(* IEC 61131-3 sources: plc/src/scl/function_blocks, 4 files *)

(* ---- dol_starter.fb ---- *)
FUNCTION_BLOCK FB DOL_Starter
VAR_INPUT
    // Digital inputs
    bStart_PB : BOOL;         // Start push button (NO)
    bStop_PB : BOOL;          // Stop push button (NC - active when pressed)
    bOverload : BOOL;         // Overload relay contact (NC - active when tripped)
    bAux_Contact : BOOL;      // Contactor auxiliary feedback (NO)
END_VAR

VAR_OUTPUT
    // Digital outputs
    bContactor : BOOL;        // Contactor coil output
    bRunning_Ind : BOOL;      // Motor running indicator
    bFault_Ind : BOOL;        // Fault indicator
    bReady_Ind : BOOL;        // Ready status indicator
END_VAR

VAR
    // Internal variables
    bLatching : BOOL;         // Latching signal
    bFault_Memory : BOOL;     // Fault memory (requires reset)
    bStart_Memory : BOOL;     // Start command memory
    bStop_Memory : BOOL;      // Stop command memory
    tStart_Delay : TON;       // Start delay timer
    tFault_Delay : TON;       // Fault delay timer
END_VAR

BEGIN
    // ==========================================
    // DOL Starter Main Control Logic
    // ==========================================

    // Input signal conditioning with debouncing
    // Rising edge detection for start button
    IF bStart_PB AND NOT bStart_Memory THEN
        bStart_Memory := TRUE;
    ELSIF NOT bStart_PB THEN
        bStart_Memory := FALSE;
    END_IF;

    // Rising edge detection for stop button (inverted - active when pressed)
    IF bStop_PB AND NOT bStop_Memory THEN
        bStop_Memory := TRUE;
    ELSIF NOT bStop_PB THEN
        bStop_Memory := FALSE;
    END_IF;

    // ==========================================
    // Main Control Circuit (Network 1 equivalent)
    // ==========================================

    // Start condition: Start button pressed AND no stop AND no overload AND no fault
    IF bStart_PB AND NOT bStop_PB AND NOT bOverload AND NOT bFault_Memory THEN
        bLatching := TRUE;
    END_IF;

    // Stop conditions: Stop button pressed OR overload OR fault
    IF bStop_PB OR bOverload OR bFault_Memory THEN
        bLatching := FALSE;
    END_IF;

    // Fault memory setting (latches fault condition)
    IF bOverload THEN
        bFault_Memory := TRUE;
    END_IF;

    // ==========================================
    // Contactor Control
    // ==========================================

    // Contactor output with latching
    // Start delay for smooth starting (optional)
    tStart_Delay(IN := bLatching, PT := T#100MS);

    bContactor := tStart_Delay.Q AND NOT bFault_Memory;

    // ==========================================
    // Status Indication (Networks 2-4 equivalent)
    // ==========================================

    // Running indicator (Network 2)
    bRunning_Ind := bContactor AND bAux_Contact;

    // Fault indicator (Network 3)
    bFault_Ind := bFault_Memory OR bOverload;

    // Ready indicator (Network 4)
    bReady_Ind := NOT bStop_PB AND NOT bOverload AND NOT bFault_Memory AND NOT bContactor;

    // ==========================================
    // Additional Safety Features
    // ==========================================

    // Contactor feedback monitoring
    // If contactor output is ON but auxiliary feedback is OFF, indicate fault
    IF bContactor AND NOT bAux_Contact THEN
        tFault_Delay(IN := TRUE, PT := T#500MS);
        IF tFault_Delay.Q THEN
            bFault_Memory := TRUE; // Contactor fault
        END_IF;
    ELSE
        tFault_Delay(IN := FALSE);
    END_IF;

    // Auto-reset fault memory when conditions are safe
    // (Optional - remove if manual reset is preferred)
    IF NOT bOverload AND NOT bContactor AND bStop_PB THEN
        // Fault can be reset by pressing stop button when safe
        bFault_Memory := FALSE;
    END_IF;

END_FUNCTION_BLOCK

(* ---- dol_starter_s7_1500.fb ---- *)
FUNCTION_BLOCK FB DOL_Starter_S7_1500
{ S7_Optimized_Access := 'TRUE' }
VAR_INPUT
    // Digital inputs
    bStart_PB : BOOL;         // Start push button (NO)
    bStop_PB : BOOL;          // Stop push button (NC - active when pressed)
    bOverload : BOOL;         // Overload relay contact (NC - active when tripped)
    bAux_Contact : BOOL;      // Contactor auxiliary feedback (NO)

    // S7-1500 specific inputs
    bEmergency_Stop : BOOL;   // Emergency stop (safety input)
    bSafety_Interlock : BOOL; // Safety interlock (safety input)
    bMaintenance_Mode : BOOL; // Maintenance mode enable
    bRemote_Enable : BOOL;    // Remote operation enable
END_VAR

VAR_OUTPUT
    // Digital outputs
    bContactor : BOOL;        // Contactor coil output
    bRunning_Ind : BOOL;      // Motor running indicator
    bFault_Ind : BOOL;        // Fault indicator
    bReady_Ind : BOOL;        // Ready status indicator

    // S7-1500 specific outputs
    bWarning_Ind : BOOL;      // Warning indicator
    bMaintenance_Ind : BOOL;   // Maintenance indicator
    bRemote_Status : BOOL;    // Remote operation status
END_VAR

VAR
    // Internal variables
    bLatching : BOOL;         // Latching signal
    bFault_Memory : BOOL;     // Fault memory (requires reset)
    bStart_Memory : BOOL;     // Start command memory
    bStop_Memory : BOOL;      // Stop command memory
    bWarning_Condition : BOOL; // Warning condition
    bStart_Command : BOOL;    // Validated start command
    bStop_Command : BOOL;     // Validated stop command

    // S7-1500 advanced timers
    tStart_Delay : TON;       // Start delay timer
    tFault_Delay : TON;       // Fault delay timer
    tWarning_Delay : TON;     // Warning delay timer
    tStartup_Delay : TON;     // Startup delay timer

    // S7-1500 specific features
    iStart_Count : DINT;      // Start counter (32-bit)
    iFault_Count : DINT;       // Fault counter (32-bit)
    rOperating_Hours : REAL;   // Operating hours (floating point)
    dtLast_Start : DT;        // Last start timestamp
    dtLast_Fault : DT;        // Last fault timestamp
    dtLast_Maintenance : DT;  // Last maintenance timestamp

    // S7-1500 diagnostic data
    bContactor_Fault : BOOL;  // Contactor fault detected
    bWiring_Fault : BOOL;     // Wiring fault detected
    bSensor_Fault : BOOL;     // Sensor fault detected
END_VAR

BEGIN
    // ==========================================
    // S7-1500 Optimized Input Processing
    // ==========================================

    // Edge detection with optimized access
    // Rising edge detection for start button
    IF bStart_PB AND NOT bStart_Memory THEN
        bStart_Memory := TRUE;
    ELSIF NOT bStart_PB THEN
        bStart_Memory := FALSE;
    END_IF;

    // Rising edge detection for stop button (inverted)
    IF bStop_PB AND NOT bStop_Memory THEN
        bStop_Memory := TRUE;
    ELSIF NOT bStop_PB THEN
        bStop_Memory := FALSE;
    END_IF;

    // ==========================================
    // S7-1500 Safety Integration
    // ==========================================

    // Emergency stop handling (priority 1)
    IF bEmergency_Stop THEN
        bContactor := FALSE;
        bFault_Memory := TRUE;
        bRunning_Ind := FALSE;
        bWarning_Condition := TRUE;
        dtLast_Fault := CURRENT_DT;
        RETURN; // Immediate exit on emergency stop
    END_IF;

    // Safety interlock handling (priority 2)
    IF bSafety_Interlock THEN
        bContactor := FALSE;
        bFault_Memory := TRUE;
        bRunning_Ind := FALSE;
        RETURN; // Immediate exit on safety interlock
    END_IF;

    // ==========================================
    // Command Validation
    // ==========================================

    // Validate start command
    bStart_Command := bStart_PB AND NOT bStop_PB AND NOT bOverload AND
                      NOT bFault_Memory AND NOT bEmergency_Stop AND NOT bSafety_Interlock;

    // Validate stop command
    bStop_Command := bStop_PB OR bOverload OR bFault_Memory;

    // ==========================================
    // S7-1500 Advanced Control Logic
    // ==========================================

    // Main control circuit with enhanced safety
    IF bStart_Command AND bRemote_Enable THEN
        bLatching := TRUE;
        iStart_Count := iStart_Count + 1;
        dtLast_Start := CURRENT_DT;
    END_IF;

    IF bStop_Command THEN
        bLatching := FALSE;
    END_IF;

    // Fault memory setting with enhanced detection
    IF bOverload OR bContactor_Fault OR bWiring_Fault OR bSensor_Fault THEN
        bFault_Memory := TRUE;
        iFault_Count := iFault_Count + 1;
        dtLast_Fault := CURRENT_DT;
    END_IF;

    // ==========================================
    // S7-1500 Enhanced Contactor Control
    // ==========================================

    // Startup delay for smooth starting
    tStartup_Delay(IN := bLatching, PT := T#200MS);

    // Start delay with optimized timing
    tStart_Delay(IN := tStartup_Delay.Q, PT := T#100MS);

    // Contactor output with safety conditions
    bContactor := tStart_Delay.Q AND NOT bFault_Memory AND
                  NOT bEmergency_Stop AND NOT bSafety_Interlock;

    // ==========================================
    // S7-1500 Advanced Diagnostics
    // ==========================================

    // Contactor feedback monitoring (S7-1500 specific)
    IF bContactor AND NOT bAux_Contact THEN
        tFault_Delay(IN := TRUE, PT := T#500MS);
        IF tFault_Delay.Q THEN
            bContactor_Fault := TRUE;
            bFault_Memory := TRUE;
        END_IF;
    ELSE
        tFault_Delay(IN := FALSE);
        bContactor_Fault := FALSE;
    END_IF;

    // Wiring fault detection
    IF bStart_PB AND bStop_PB THEN
        bWiring_Fault := TRUE;
        bFault_Memory := TRUE;
    ELSE
        bWiring_Fault := FALSE;
    END_IF;

    // ==========================================
    // S7-1500 Enhanced Status Indication
    // ==========================================

    // Running indicator with feedback verification
    bRunning_Ind := bContactor AND bAux_Contact AND NOT bFault_Memory;

    // Fault indicator with multiple fault sources
    bFault_Ind := bFault_Memory OR bOverload OR bContactor_Fault OR
                  bWiring_Fault OR bSensor_Fault;

    // Ready indicator with comprehensive conditions
    bReady_Ind := NOT bStop_PB AND NOT bOverload AND NOT bFault_Memory AND
                  NOT bContactor AND NOT bEmergency_Stop AND NOT bSafety_Interlock;

    // Warning indicator for predictive maintenance
    tWarning_Delay(IN := (iStart_Count > 10000) OR (rOperating_Hours > 10000.0),
                   PT := T#5S);
    bWarning_Ind := tWarning_Delay.Q OR bWarning_Condition;

    // Maintenance indicator
    bMaintenance_Ind := bMaintenance_Mode;

    // Remote status indicator
    bRemote_Status := bRemote_Enable;

    // ==========================================
    // S7-1500 Operating Hours Calculation
    // ==========================================

    // Calculate operating hours (increment every cycle when running)
    IF bRunning_Ind THEN
        rOperating_Hours := rOperating_Hours + 0.0001; // Approximate per cycle
    END_IF;

    // ==========================================
    // S7-1500 Enhanced Fault Reset
    // ==========================================

    // Enhanced fault reset with safety conditions
    IF NOT bOverload AND NOT bContactor_Fault AND NOT bWiring_Fault AND
       NOT bSensor_Fault AND NOT bContactor AND bStop_PB AND bMaintenance_Mode THEN
        // Fault can be reset in maintenance mode
        bFault_Memory := FALSE;
        bWarning_Condition := FALSE;
        dtLast_Maintenance := CURRENT_DT;
    END_IF;

END_FUNCTION_BLOCK

(* ---- dol_starter_test.fb ---- *)
FUNCTION_BLOCK FB DOL_Starter_Test
VAR_INPUT
    // Test control inputs
    bTest_Mode_Enable : BOOL;     // Enable test mode
    bTest_Start_PB : BOOL;        // Test start button simulation
    bTest_Stop_PB : BOOL;         // Test stop button simulation
    bTest_Overload : BOOL;        // Test overload simulation
    bTest_Contactor_FB : BOOL;    // Test contactor feedback simulation
    bManual_Contactor_Test : BOOL; // Manual contactor test
    bReset_Test : BOOL;           // Reset test results
END_VAR

VAR_OUTPUT
    // Simulated outputs to DOL starter
    bSim_Start_PB : BOOL;         // Simulated start to DOL starter
    bSim_Stop_PB : BOOL;          // Simulated stop to DOL starter
    bSim_Overload : BOOL;         // Simulated overload to DOL starter
    bSim_Aux_Contact : BOOL;      // Simulated aux contact to DOL starter
    bTest_Mode_Active : BOOL;     // Test mode indicator
    bTest_Contactor_Out : BOOL;   // Manual test contactor output

    // Test verification outputs
    bRunning_Verified : BOOL;     // Running status verified
    bFault_Verified : BOOL;       // Fault status verified
    bReady_Verified : BOOL;       // Ready status verified
    bTest_Success : BOOL;         // Test passed indication
    bTest_Fail : BOOL;            // Test failed indication
END_VAR

VAR_IN_OUT
    // Connection to DOL starter
    bDOL_Contactor : BOOL;        // DOL starter contactor output
    bDOL_Running_Ind : BOOL;      // DOL starter running indicator
    bDOL_Fault_Ind : BOOL;        // DOL starter fault indicator
    bDOL_Ready_Ind : BOOL;        // DOL starter ready indicator
END_VAR

VAR
    // Internal test variables
    bTest_Result_Latch : BOOL;    // Test result latch
    bStart_Test_Pass : BOOL;       // Start test pass flag
    bStop_Test_Pass : BOOL;        // Stop test pass flag
    bOverload_Test_Pass : BOOL;    // Overload test pass flag
    bFeedback_Test_Pass : BOOL;   // Feedback test pass flag
    iTest_Counter : INT;           // Test counter
    tTest_Delay : TON;             // Test delay timer
END_VAR

BEGIN
    // ==========================================
    // Test Mode Control
    // ==========================================

    bTest_Mode_Active := bTest_Mode_Enable;

    // Reset test results
    IF bReset_Test THEN
        bTest_Result_Latch := FALSE;
        bTest_Success := FALSE;
        bTest_Fail := FALSE;
        bStart_Test_Pass := FALSE;
        bStop_Test_Pass := FALSE;
        bOverload_Test_Pass := FALSE;
        bFeedback_Test_Pass := FALSE;
        iTest_Counter := 0;
    END_IF;

    // ==========================================
    // Signal Simulation (when test mode enabled)
    // ==========================================

    IF bTest_Mode_Enable THEN
        // Simulate inputs to DOL starter
        bSim_Start_PB := bTest_Start_PB;
        bSim_Stop_PB := bTest_Stop_PB;
        bSim_Overload := bTest_Overload;
        bSim_Aux_Contact := bTest_Contactor_FB OR bDOL_Contactor;

        // Manual contactor test
        bTest_Contactor_Out := bManual_Contactor_Test;
    ELSE
        // Pass through real signals when not in test mode
        bSim_Start_PB := FALSE;  // Disable simulation
        bSim_Stop_PB := FALSE;
        bSim_Overload := FALSE;
        bSim_Aux_Contact := bDOL_Contactor;
        bTest_Contactor_Out := FALSE;
    END_IF;

    // ==========================================
    // Test Verification Logic
    // ==========================================

    // Running status verification
    // Contact output ON and running indicator ON = verified
    bRunning_Verified := bDOL_Contactor AND bDOL_Running_Ind;

    // Fault status verification
    // Fault indicator ON or overload active = verified
    bFault_Verified := bDOL_Fault_Ind OR bSim_Overload;

    // Ready status verification
    // No stop, no overload, no contactor = ready
    bReady_Verified := NOT bSim_Stop_PB AND NOT bSim_Overload AND NOT bDOL_Contactor;

    // ==========================================
    // Automated Test Sequences
    // ==========================================

    // Test 1: Start Button Test
    IF bTest_Start_PB AND NOT bStart_Test_Pass AND bTest_Mode_Enable THEN
        tTest_Delay(IN := TRUE, PT := T#500MS);
        IF tTest_Delay.Q AND bDOL_Contactor AND bDOL_Running_Ind THEN
            bStart_Test_Pass := TRUE;
            iTest_Counter := iTest_Counter + 1;
        END_IF;
    ELSE
        tTest_Delay(IN := FALSE);
    END_IF;

    // Test 2: Stop Button Test
    IF bTest_Stop_PB AND NOT bStop_Test_Pass AND bTest_Mode_Enable THEN
        tTest_Delay(IN := TRUE, PT := T#500MS);
        IF tTest_Delay.Q AND NOT bDOL_Contactor AND NOT bDOL_Running_Ind AND bDOL_Ready_Ind THEN
            bStop_Test_Pass := TRUE;
            iTest_Counter := iTest_Counter + 1;
        END_IF;
    ELSE
        tTest_Delay(IN := FALSE);
    END_IF;

    // Test 3: Overload Test
    IF bTest_Overload AND NOT bOverload_Test_Pass AND bTest_Mode_Enable THEN
        tTest_Delay(IN := TRUE, PT := T#500MS);
        IF tTest_Delay.Q AND NOT bDOL_Contactor AND bDOL_Fault_Ind THEN
            bOverload_Test_Pass := TRUE;
            iTest_Counter := iTest_Counter + 1;
        END_IF;
    ELSE
        tTest_Delay(IN := FALSE);
    END_IF;

    // Test 4: Contactor Feedback Test
    IF bTest_Contactor_FB AND NOT bFeedback_Test_Pass AND bTest_Mode_Enable THEN
        tTest_Delay(IN := TRUE, PT := T#1S);
        IF tTest_Delay.Q AND bDOL_Fault_Ind THEN
            bFeedback_Test_Pass := TRUE;
            iTest_Counter := iTest_Counter + 1;
        END_IF;
    ELSE
        tTest_Delay(IN := FALSE);
    END_IF;

    // ==========================================
    // Test Result Evaluation
    // ==========================================

    // Overall test result
    IF bStart_Test_Pass AND bStop_Test_Pass AND bOverload_Test_Pass AND bFeedback_Test_Pass THEN
        bTest_Success := TRUE;
        bTest_Fail := FALSE;
        bTest_Result_Latch := TRUE;
    ELSIF (bTest_Start_PB OR bTest_Stop_PB OR bTest_Overload OR bTest_Contactor_FB) AND
           NOT (bStart_Test_Pass AND bStop_Test_Pass AND bOverload_Test_Pass AND bFeedback_Test_Pass) THEN
        // Individual test failures
        IF NOT bStart_Test_Pass AND bTest_Start_PB THEN
            bTest_Fail := TRUE;
        END_IF;
        IF NOT bStop_Test_Pass AND bTest_Stop_PB THEN
            bTest_Fail := TRUE;
        END_IF;
        IF NOT bOverload_Test_Pass AND bTest_Overload THEN
            bTest_Fail := TRUE;
        END_IF;
        IF NOT bFeedback_Test_Pass AND bTest_Contactor_FB THEN
            bTest_Fail := TRUE;
        END_IF;
    END_IF;

END_FUNCTION_BLOCK

(* ---- motor_control.fb ---- *)
FUNCTION_BLOCK FB Motor_Control
VAR_INPUT
    // Motor control inputs
    bStart : BOOL;         // Start command
    bStop : BOOL;          // Stop command
    bEmergency : BOOL;     // Emergency stop
    bAutoMode : BOOL;      // Automatic mode
    rSpeedSetpoint : REAL; // Speed setpoint (0-100%)
END_VAR

VAR_OUTPUT
    // Motor control outputs
    bRun : BOOL;           // Motor running
    bFault : BOOL;         // Fault condition
    rActualSpeed : REAL;   // Actual speed feedback
    bReady : BOOL;         // Ready for operation
END_VAR

VAR
    // Internal variables
    tTimer : TON;          // Timer for startup
    rCurrentSpeed : REAL;  // Internal speed variable
    bFaultCondition : BOOL; // Internal fault flag
END_VAR

BEGIN
    // Emergency stop handling
    IF bEmergency THEN
        bRun := FALSE;
        bFault := TRUE;
        rCurrentSpeed := 0.0;
        rActualSpeed := 0.0;
        bReady := FALSE;
        RETURN;
    END_IF;

    // Stop command handling
    IF bStop THEN
        bRun := FALSE;
        rCurrentSpeed := 0.0;
        rActualSpeed := 0.0;
        bReady := TRUE;
        RETURN;
    END_IF;

    // Start command handling
    IF bStart AND NOT bFault THEN
        bRun := TRUE;
        bReady := FALSE;

        // Speed control
        IF bAutoMode THEN
            // Automatic speed control
            IF rCurrentSpeed < rSpeedSetpoint THEN
                rCurrentSpeed := rCurrentSpeed + 1.0;
            ELSIF rCurrentSpeed > rSpeedSetpoint THEN
                rCurrentSpeed := rCurrentSpeed - 1.0;
            END_IF;
        ELSE
            // Manual speed control
            rCurrentSpeed := rSpeedSetpoint;
        END_IF;

        rActualSpeed := rCurrentSpeed;

        // Check for fault conditions
        IF rActualSpeed < 0.0 OR rActualSpeed > 100.0 THEN
            bFault := TRUE;
            bRun := FALSE;
        END_IF;
    ELSE
        bRun := FALSE;
        rCurrentSpeed := 0.0;
        rActualSpeed := 0.0;
        bReady := TRUE;
    END_IF;
END_FUNCTION_BLOCK
